// TIA Portal V17 export
// export: Created 2025-07-01T09:58:23.6431093Z, ExportSetting WithDefaults, DisplayName Totally Integrated Automation Portal, DisplayVersion V17 Update 8, DisplayName TIA Portal Openness, DisplayVersion V17 Update 8, DisplayName TIA Portal Version Control Interface, DisplayVersion V17, DisplayName SINAMICS Startdrive Advanced, DisplayVersion V17 SP2, DisplayName SINAMICS Startdrive G110M, G120, G120C, G120D, G120P, G115D, DisplayVersion V17 SP2, DisplayName SINAMICS Startdrive G130, G150, S120, S150, SINAMICS MV, S210, DisplayVersion V17 SP2, DisplayName STEP 7 Professional, DisplayVersion V17 Update 8, DisplayName SINUMERIK ONE STEP 7 Toolbox, DisplayVersion V17 Update 12, DisplayName SINUMERIK ONE PLC Basic Program Plus, DisplayVersion V17 Update 12, DisplayName SINUMERIK 840D sl STEP 7 Toolbox, DisplayVersion V17 Update 12, DisplayName STEP 7 Safety, DisplayVersion V17 Update 6, DisplayName WinCC Advanced, DisplayVersion V17 Update 8
FUNCTION_BLOCK "FB10400_PRESSURE_SENSOR"   // FB10400, LAD
{ S7_Optimized_Access := 'FALSE' }
VERSION : 0.1
// stored: AutoNumber false, IsIECCheckEnabled false, SetENOAutomatically false, UDAEnableTagReadback false
   VAR_INPUT
      SENSOR_VALUE_I : Int;   // SENSOR VALUE INPUT
      STATION_CYCLE_RUNNING : Bool;   // STATION CYCLE RUNNING
   END_VAR
   VAR_OUTPUT
      LOW_PRESSURE_ALARM : Bool;   // ASPIRATION PRESSURE TOO LOW ALARM
      HIGH_PRESSURE_ALARM : Bool;   // ASPIRATION PRESSURE TOO HIGH ALARM
      LOW_PRESSURE_WARNING : Bool;   // ASPIRATION PRESSURE TOO LOW WARNING
      HIGH_PRESSURE_WARNING : Bool;   // ASPIRATION PRESSURE TOO HIGH WARNING
   END_VAR
   VAR DB_SPECIFIC
      HMI : Struct
         HIGH_LIMIT_ALARM_VALUE : Real;   // HIGH LIMIT ALARM VALUE
         HIGH_LIMIT_WARNING_VALUE : Real;   // HIGH LIMIT WARNING VALUE
         LOW_LIMIT_ALARM_VALUE : Real;   // LOW LIMIT ALARM VALUE
         LOW_LIMIT_WARNING_VALUE : Real;   // LOW LIMIT WARNING VALUE
      END_STRUCT;
      SETTINGS : Struct
         NORM_MIN_VAL : Int;   // NORMALIZE MIN VALUE
         NORM_MAX_VAL : Int;   // NORMALIZE MAX VALUE
         SCALE_MIN_VAL : Real;   // SCALE MIN VALUE
         SCALE_MAX_VAL : Real;   // SCALE MAX VALUE
         MUL_VAL : Real;   // MULTIPLY VALUE
         DIV_VAL : Real;   // DIVIDE VALUE
         UNIT_NO : Int;   // UNIT NUMBER
      END_STRUCT;
      OUTPUT : Struct
         PRESSURE_VALUE : Real;   // PRESSURE VALUE
      END_STRUCT;
      INTERNAL : Struct
         NORMALIZED_VALUE : Real;   // NORMALIZED VALUE
         SCALED_VALUE : Real;   // SCALED VALUE
         MULTIPLIED_VALUE : Real;   // MULTIPLIED VALUE
      END_STRUCT;
      ALARMS : Struct
         LOW_PRESSURE_ALARM : Bool;   // ASPIRATION PRESSURE TOO LOW ALARM
         HIGH_PRESSURE_ALARM : Bool;   // ASPIRATION PRESSURE TOO HIGH ALARM
         LOW_PRESSURE_WARNING : Bool;   // ASPIRATION PRESSURE TOO LOW WARNING
         HIGH_PRESSURE_WARNING : Bool;   // ASPIRATION PRESSURE TOO HIGH WARNING
      END_STRUCT;
      TIMERS : Struct
         ASPIRATION_LOW_ALARM_TIMER : TON_TIME;
         ASPIRATION_LOW_WARNING_TIMER : TON_TIME;
         ASPIRATION_HIGH_ALARM_TIMER : TON_TIME;
         ASPIRATION_HIGH_WARNING_TIMER : TON_TIME;
      END_STRUCT;
   END_VAR
   VAR_TEMP
      DB_NUMBER : DInt;   // DB NUMBER
   END_VAR
   VAR_TEMP   // added for the SCL form of the ladder/FBD networks
      _w1 : Bool;
   END_VAR
BEGIN

NETWORK
TITLE = READ INSTANCE DB
      L     DINO;
      +     10#800000;
      T     #DB_NUMBER;


REGION Network 2: PRESSURE VALUE
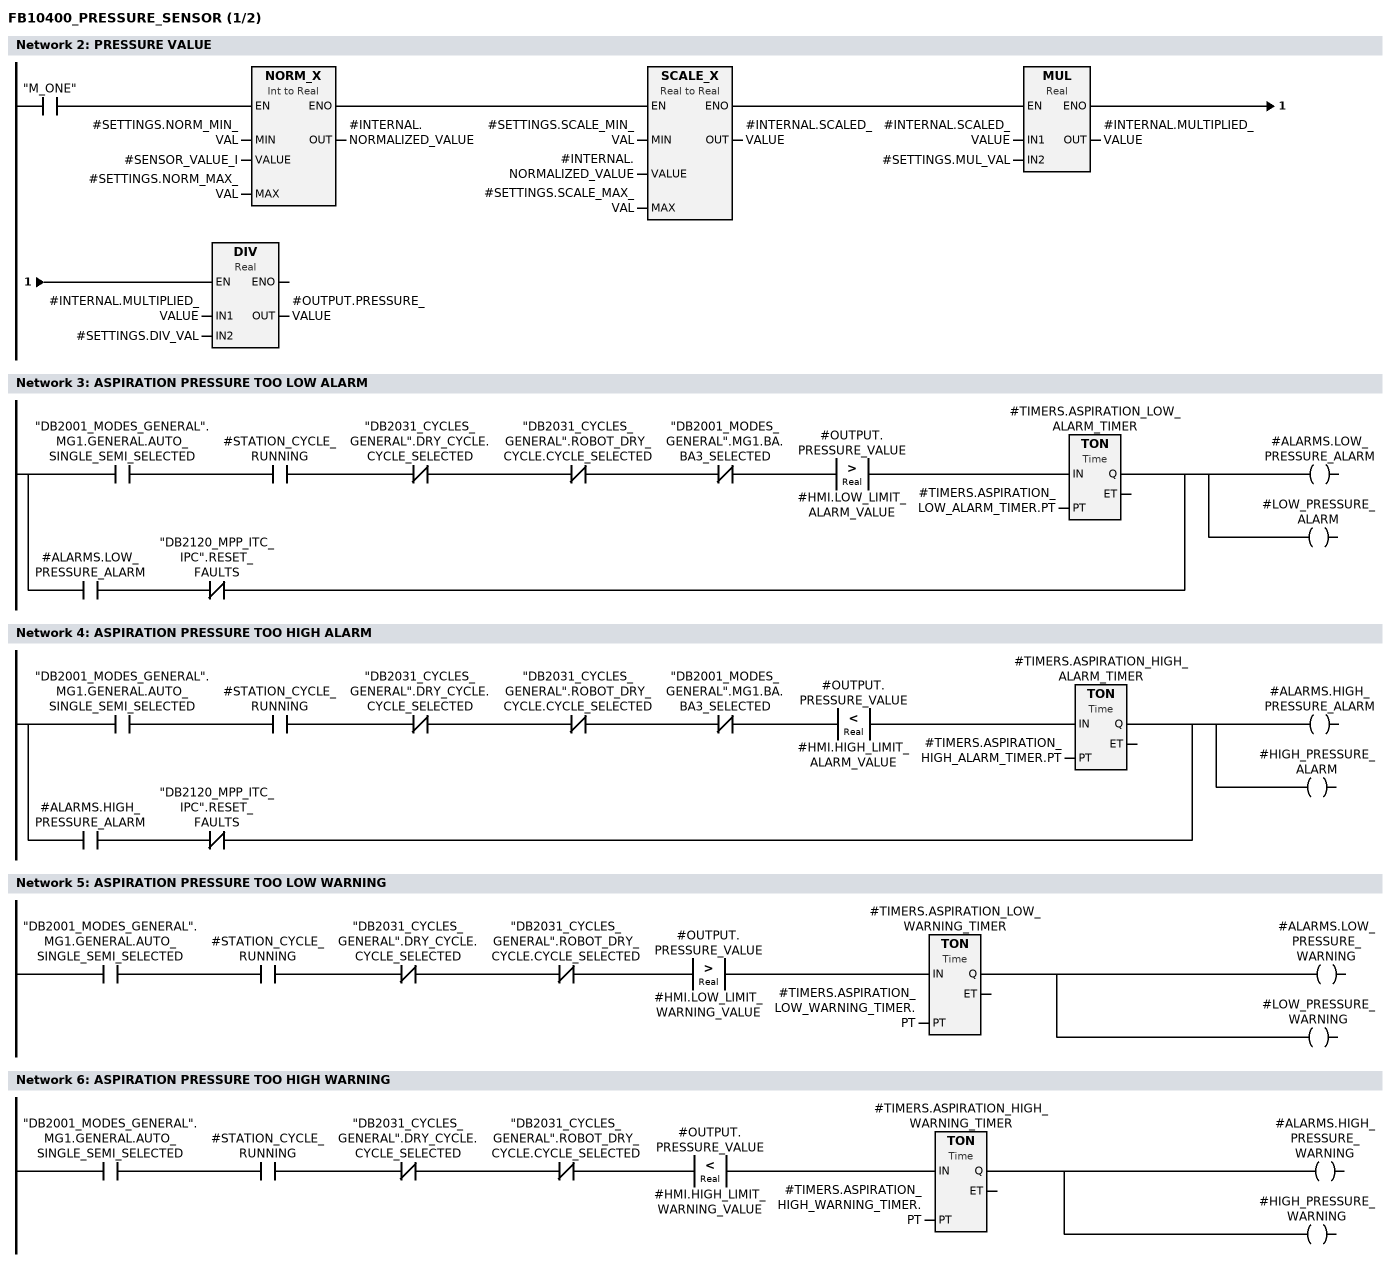
   RUNG wire#powerrail
      Contact( "M_ONE" )
      { S7_Templates := "[SrcType := Int, DestType := Real]" } Normalize(min := #SETTINGS.NORM_MIN_VAL, value := #SENSOR_VALUE_I, max := #SETTINGS.NORM_MAX_VAL, out => #INTERNAL.NORMALIZED_VALUE)
      { S7_Templates := "[SrcType := Real, DestType := Real]" } Scale(min := #SETTINGS.SCALE_MIN_VAL, value := #INTERNAL.NORMALIZED_VALUE, max := #SETTINGS.SCALE_MAX_VAL, out => #INTERNAL.SCALED_VALUE)
      { S7_Templates := "SrcType := Real" } Mul(in1 := #INTERNAL.SCALED_VALUE, in2 := #SETTINGS.MUL_VAL, out => #INTERNAL.MULTIPLIED_VALUE)
      { S7_Templates := "SrcType := Real" } Div(in1 := #INTERNAL.MULTIPLIED_VALUE, in2 := #SETTINGS.DIV_VAL, out => #OUTPUT.PRESSURE_VALUE)
   END_RUNG
   // the same network as SCL:
   IF "M_ONE" THEN
       #INTERNAL.NORMALIZED_VALUE := NORM_X(MIN := #SETTINGS.NORM_MIN_VAL, VALUE := #SENSOR_VALUE_I, MAX := #SETTINGS.NORM_MAX_VAL);
       #INTERNAL.SCALED_VALUE := SCALE_X(MIN := #SETTINGS.SCALE_MIN_VAL, VALUE := #INTERNAL.NORMALIZED_VALUE, MAX := #SETTINGS.SCALE_MAX_VAL);
       #INTERNAL.MULTIPLIED_VALUE := #INTERNAL.SCALED_VALUE * #SETTINGS.MUL_VAL;
       #OUTPUT.PRESSURE_VALUE := #INTERNAL.MULTIPLIED_VALUE / #SETTINGS.DIV_VAL;
   END_IF;
END_REGION

REGION Network 3: ASPIRATION PRESSURE TOO LOW ALARM
   RUNG wire#powerrail
      Contact( "DB2001_MODES_GENERAL".MG1.GENERAL.AUTO_SINGLE_SEMI_SELECTED )
      Contact( #STATION_CYCLE_RUNNING )
      I_Contact( "DB2031_CYCLES_GENERAL".DRY_CYCLE.CYCLE_SELECTED )
      I_Contact( "DB2031_CYCLES_GENERAL".ROBOT_DRY_CYCLE.CYCLE_SELECTED )
      I_Contact( "DB2001_MODES_GENERAL".MG1.BA.BA3_SELECTED )
      { S7_Templates := "SrcType := Real" } GT_Contact(in1 := #OUTPUT.PRESSURE_VALUE, in2 := #HMI.LOW_LIMIT_ALARM_VALUE)
      { S7_Templates := "time_type := Time" } #TIMERS.ASPIRATION_LOW_ALARM_TIMER.TON(pt := #TIMERS.ASPIRATION_LOW_ALARM_TIMER.PT, et =>)
      wire#w1
      Coil( #ALARMS.LOW_PRESSURE_ALARM )
   END_RUNG
   RUNG wire#powerrail
      Contact( #ALARMS.LOW_PRESSURE_ALARM )
      I_Contact( "DB2120_MPP_ITC_IPC".RESET_FAULTS )
   END_RUNG wire#w1
   RUNG wire#w1
      Coil( #LOW_PRESSURE_ALARM )
   END_RUNG
   // the same network as SCL:
   #TIMERS.ASPIRATION_LOW_ALARM_TIMER.TON(IN := "DB2001_MODES_GENERAL".MG1.GENERAL.AUTO_SINGLE_SEMI_SELECTED AND #STATION_CYCLE_RUNNING AND NOT "DB2031_CYCLES_GENERAL".DRY_CYCLE.CYCLE_SELECTED AND NOT "DB2031_CYCLES_GENERAL".ROBOT_DRY_CYCLE.CYCLE_SELECTED AND NOT "DB2001_MODES_GENERAL".MG1.BA.BA3_SELECTED AND (#OUTPUT.PRESSURE_VALUE > #HMI.LOW_LIMIT_ALARM_VALUE),
                           PT := #TIMERS.ASPIRATION_LOW_ALARM_TIMER.PT);
   #ALARMS.LOW_PRESSURE_ALARM := #TIMERS.ASPIRATION_LOW_ALARM_TIMER.Q OR (#ALARMS.LOW_PRESSURE_ALARM AND NOT "DB2120_MPP_ITC_IPC".RESET_FAULTS);
   #LOW_PRESSURE_ALARM := #ALARMS.LOW_PRESSURE_ALARM;
END_REGION

REGION Network 4: ASPIRATION PRESSURE TOO HIGH ALARM
   RUNG wire#powerrail
      Contact( "DB2001_MODES_GENERAL".MG1.GENERAL.AUTO_SINGLE_SEMI_SELECTED )
      Contact( #STATION_CYCLE_RUNNING )
      I_Contact( "DB2031_CYCLES_GENERAL".DRY_CYCLE.CYCLE_SELECTED )
      I_Contact( "DB2031_CYCLES_GENERAL".ROBOT_DRY_CYCLE.CYCLE_SELECTED )
      I_Contact( "DB2001_MODES_GENERAL".MG1.BA.BA3_SELECTED )
      { S7_Templates := "SrcType := Real" } LT_Contact(in1 := #OUTPUT.PRESSURE_VALUE, in2 := #HMI.HIGH_LIMIT_ALARM_VALUE)
      { S7_Templates := "time_type := Time" } #TIMERS.ASPIRATION_HIGH_ALARM_TIMER.TON(pt := #TIMERS.ASPIRATION_HIGH_ALARM_TIMER.PT, et =>)
      wire#w1
      Coil( #ALARMS.HIGH_PRESSURE_ALARM )
   END_RUNG
   RUNG wire#powerrail
      Contact( #ALARMS.HIGH_PRESSURE_ALARM )
      I_Contact( "DB2120_MPP_ITC_IPC".RESET_FAULTS )
   END_RUNG wire#w1
   RUNG wire#w1
      Coil( #HIGH_PRESSURE_ALARM )
   END_RUNG
   // the same network as SCL:
   #TIMERS.ASPIRATION_HIGH_ALARM_TIMER.TON(IN := "DB2001_MODES_GENERAL".MG1.GENERAL.AUTO_SINGLE_SEMI_SELECTED AND #STATION_CYCLE_RUNNING AND NOT "DB2031_CYCLES_GENERAL".DRY_CYCLE.CYCLE_SELECTED AND NOT "DB2031_CYCLES_GENERAL".ROBOT_DRY_CYCLE.CYCLE_SELECTED AND NOT "DB2001_MODES_GENERAL".MG1.BA.BA3_SELECTED AND (#OUTPUT.PRESSURE_VALUE < #HMI.HIGH_LIMIT_ALARM_VALUE),
                           PT := #TIMERS.ASPIRATION_HIGH_ALARM_TIMER.PT);
   #ALARMS.HIGH_PRESSURE_ALARM := #TIMERS.ASPIRATION_HIGH_ALARM_TIMER.Q OR (#ALARMS.HIGH_PRESSURE_ALARM AND NOT "DB2120_MPP_ITC_IPC".RESET_FAULTS);
   #HIGH_PRESSURE_ALARM := #ALARMS.HIGH_PRESSURE_ALARM;
END_REGION

REGION Network 5: ASPIRATION PRESSURE TOO LOW WARNING
   RUNG wire#powerrail
      Contact( "DB2001_MODES_GENERAL".MG1.GENERAL.AUTO_SINGLE_SEMI_SELECTED )
      Contact( #STATION_CYCLE_RUNNING )
      I_Contact( "DB2031_CYCLES_GENERAL".DRY_CYCLE.CYCLE_SELECTED )
      I_Contact( "DB2031_CYCLES_GENERAL".ROBOT_DRY_CYCLE.CYCLE_SELECTED )
      { S7_Templates := "SrcType := Real" } GT_Contact(in1 := #OUTPUT.PRESSURE_VALUE, in2 := #HMI.LOW_LIMIT_WARNING_VALUE)
      { S7_Templates := "time_type := Time" } #TIMERS.ASPIRATION_LOW_WARNING_TIMER.TON(pt := #TIMERS.ASPIRATION_LOW_WARNING_TIMER.PT, et =>)
      wire#w1
      Coil( #ALARMS.LOW_PRESSURE_WARNING )
   END_RUNG
   RUNG wire#w1
      Coil( #LOW_PRESSURE_WARNING )
   END_RUNG
   // the same network as SCL:
   #TIMERS.ASPIRATION_LOW_WARNING_TIMER.TON(IN := "DB2001_MODES_GENERAL".MG1.GENERAL.AUTO_SINGLE_SEMI_SELECTED AND #STATION_CYCLE_RUNNING AND NOT "DB2031_CYCLES_GENERAL".DRY_CYCLE.CYCLE_SELECTED AND NOT "DB2031_CYCLES_GENERAL".ROBOT_DRY_CYCLE.CYCLE_SELECTED AND (#OUTPUT.PRESSURE_VALUE > #HMI.LOW_LIMIT_WARNING_VALUE),
                           PT := #TIMERS.ASPIRATION_LOW_WARNING_TIMER.PT);
   #ALARMS.LOW_PRESSURE_WARNING := #TIMERS.ASPIRATION_LOW_WARNING_TIMER.Q;
   #LOW_PRESSURE_WARNING := #TIMERS.ASPIRATION_LOW_WARNING_TIMER.Q;
END_REGION

REGION Network 6: ASPIRATION PRESSURE TOO HIGH WARNING
   RUNG wire#powerrail
      Contact( "DB2001_MODES_GENERAL".MG1.GENERAL.AUTO_SINGLE_SEMI_SELECTED )
      Contact( #STATION_CYCLE_RUNNING )
      I_Contact( "DB2031_CYCLES_GENERAL".DRY_CYCLE.CYCLE_SELECTED )
      I_Contact( "DB2031_CYCLES_GENERAL".ROBOT_DRY_CYCLE.CYCLE_SELECTED )
      { S7_Templates := "SrcType := Real" } LT_Contact(in1 := #OUTPUT.PRESSURE_VALUE, in2 := #HMI.HIGH_LIMIT_WARNING_VALUE)
      { S7_Templates := "time_type := Time" } #TIMERS.ASPIRATION_HIGH_WARNING_TIMER.TON(pt := #TIMERS.ASPIRATION_HIGH_WARNING_TIMER.PT, et =>)
      wire#w1
      Coil( #ALARMS.HIGH_PRESSURE_WARNING )
   END_RUNG
   RUNG wire#w1
      Coil( #HIGH_PRESSURE_WARNING )
   END_RUNG
   // the same network as SCL:
   #TIMERS.ASPIRATION_HIGH_WARNING_TIMER.TON(IN := "DB2001_MODES_GENERAL".MG1.GENERAL.AUTO_SINGLE_SEMI_SELECTED AND #STATION_CYCLE_RUNNING AND NOT "DB2031_CYCLES_GENERAL".DRY_CYCLE.CYCLE_SELECTED AND NOT "DB2031_CYCLES_GENERAL".ROBOT_DRY_CYCLE.CYCLE_SELECTED AND (#OUTPUT.PRESSURE_VALUE < #HMI.HIGH_LIMIT_WARNING_VALUE),
                           PT := #TIMERS.ASPIRATION_HIGH_WARNING_TIMER.PT);
   #ALARMS.HIGH_PRESSURE_WARNING := #TIMERS.ASPIRATION_HIGH_WARNING_TIMER.Q;
   #HIGH_PRESSURE_WARNING := #TIMERS.ASPIRATION_HIGH_WARNING_TIMER.Q;
END_REGION

REGION Network 7: IMMEDIATE STOP AND STOP END OF CYCLE ALARMS
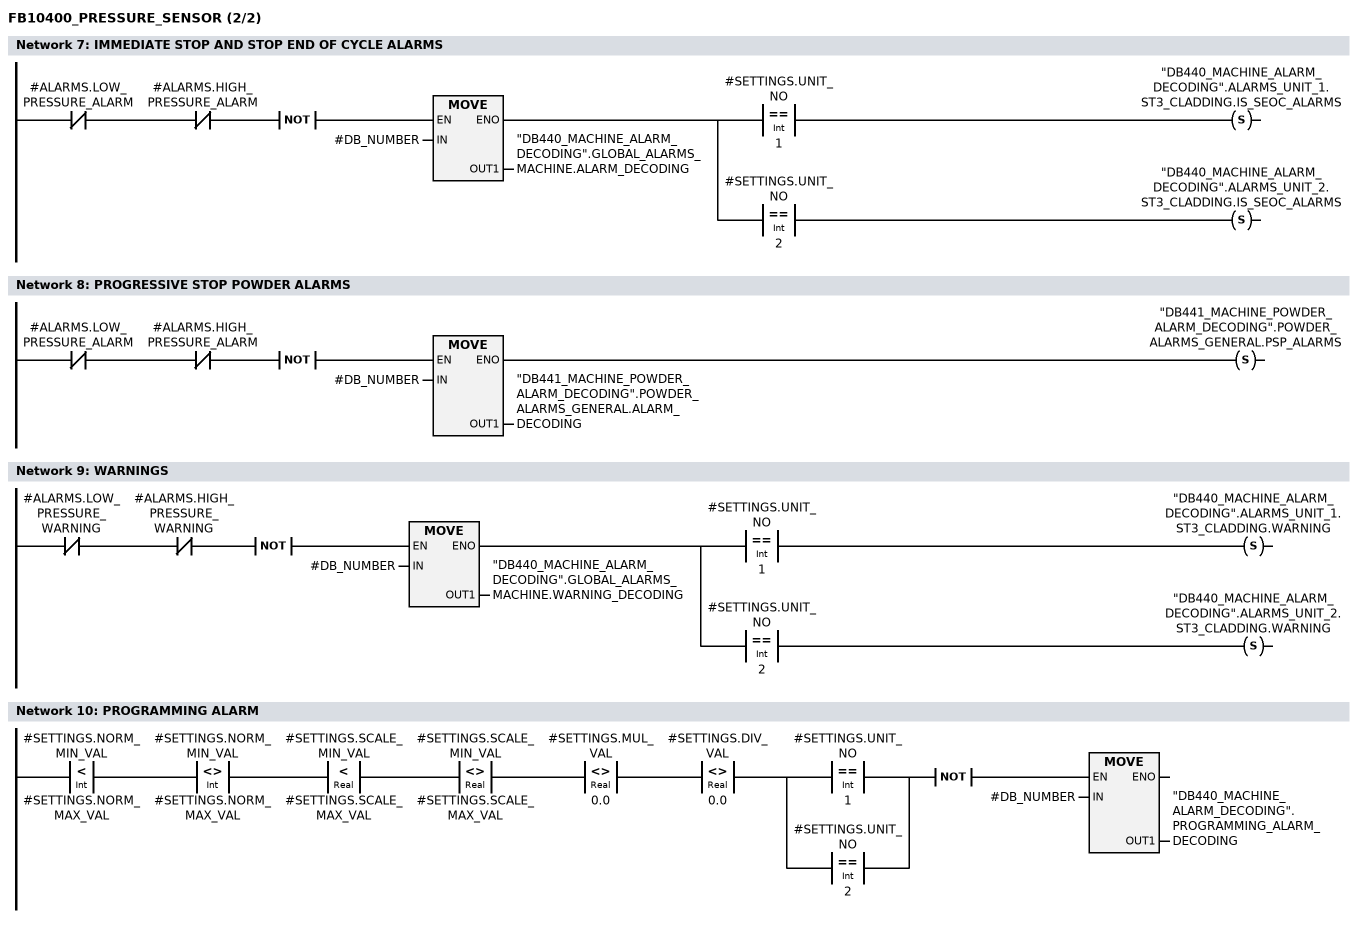
   RUNG wire#powerrail
      I_Contact( #ALARMS.LOW_PRESSURE_ALARM )
      I_Contact( #ALARMS.HIGH_PRESSURE_ALARM )
      Not()
      { S7_GenerateENO := "TRUE" } Move(in := #DB_NUMBER, out1 => "DB440_MACHINE_ALARM_DECODING".GLOBAL_ALARMS_MACHINE.ALARM_DECODING)
      wire#w1
      { S7_Templates := "SrcType := Int" } EQ_Contact(in1 := #SETTINGS.UNIT_NO, in2 := 1)
      S_Coil( "DB440_MACHINE_ALARM_DECODING".ALARMS_UNIT_1.ST3_CLADDING.IS_SEOC_ALARMS )
   END_RUNG
   RUNG wire#w1
      { S7_Templates := "SrcType := Int" } EQ_Contact(in1 := #SETTINGS.UNIT_NO, in2 := 2)
      S_Coil( "DB440_MACHINE_ALARM_DECODING".ALARMS_UNIT_2.ST3_CLADDING.IS_SEOC_ALARMS )
   END_RUNG
   // the same network as SCL:
   // ENO of a box is taken as its EN; it also drops when the box reports an error
   #_w1 := NOT (NOT #ALARMS.LOW_PRESSURE_ALARM AND NOT #ALARMS.HIGH_PRESSURE_ALARM);
   IF #_w1 THEN "DB440_MACHINE_ALARM_DECODING".GLOBAL_ALARMS_MACHINE.ALARM_DECODING := #DB_NUMBER; END_IF;
   IF #_w1 AND (#SETTINGS.UNIT_NO = 1) THEN
       "DB440_MACHINE_ALARM_DECODING".ALARMS_UNIT_1.ST3_CLADDING.IS_SEOC_ALARMS := TRUE;
   END_IF;
   IF #_w1 AND (#SETTINGS.UNIT_NO = 2) THEN
       "DB440_MACHINE_ALARM_DECODING".ALARMS_UNIT_2.ST3_CLADDING.IS_SEOC_ALARMS := TRUE;
   END_IF;
END_REGION

REGION Network 8: PROGRESSIVE STOP POWDER ALARMS
   RUNG wire#powerrail
      I_Contact( #ALARMS.LOW_PRESSURE_ALARM )
      I_Contact( #ALARMS.HIGH_PRESSURE_ALARM )
      Not()
      { S7_GenerateENO := "TRUE" } Move(in := #DB_NUMBER, out1 => "DB441_MACHINE_POWDER_ALARM_DECODING".POWDER_ALARMS_GENERAL.ALARM_DECODING)
      S_Coil( "DB441_MACHINE_POWDER_ALARM_DECODING".POWDER_ALARMS_GENERAL.PSP_ALARMS )
   END_RUNG
   // the same network as SCL:
   // ENO of a box is taken as its EN; it also drops when the box reports an error
   IF NOT (NOT #ALARMS.LOW_PRESSURE_ALARM AND NOT #ALARMS.HIGH_PRESSURE_ALARM) THEN
       "DB441_MACHINE_POWDER_ALARM_DECODING".POWDER_ALARMS_GENERAL.ALARM_DECODING := #DB_NUMBER;
       "DB441_MACHINE_POWDER_ALARM_DECODING".POWDER_ALARMS_GENERAL.PSP_ALARMS := TRUE;
   END_IF;
END_REGION

REGION Network 9: WARNINGS
   RUNG wire#powerrail
      I_Contact( #ALARMS.LOW_PRESSURE_WARNING )
      I_Contact( #ALARMS.HIGH_PRESSURE_WARNING )
      Not()
      Move(in := #DB_NUMBER, out1 => "DB440_MACHINE_ALARM_DECODING".GLOBAL_ALARMS_MACHINE.WARNING_DECODING)
      wire#w1
      { S7_Templates := "SrcType := Int" } EQ_Contact(in1 := #SETTINGS.UNIT_NO, in2 := 1)
      S_Coil( "DB440_MACHINE_ALARM_DECODING".ALARMS_UNIT_1.ST3_CLADDING.WARNING )
   END_RUNG
   RUNG wire#w1
      { S7_Templates := "SrcType := Int" } EQ_Contact(in1 := #SETTINGS.UNIT_NO, in2 := 2)
      S_Coil( "DB440_MACHINE_ALARM_DECODING".ALARMS_UNIT_2.ST3_CLADDING.WARNING )
   END_RUNG
   // the same network as SCL:
   #_w1 := NOT (NOT #ALARMS.LOW_PRESSURE_WARNING AND NOT #ALARMS.HIGH_PRESSURE_WARNING);
   IF #_w1 THEN "DB440_MACHINE_ALARM_DECODING".GLOBAL_ALARMS_MACHINE.WARNING_DECODING := #DB_NUMBER; END_IF;
   IF #_w1 AND (#SETTINGS.UNIT_NO = 1) THEN
       "DB440_MACHINE_ALARM_DECODING".ALARMS_UNIT_1.ST3_CLADDING.WARNING := TRUE;
   END_IF;
   IF #_w1 AND (#SETTINGS.UNIT_NO = 2) THEN
       "DB440_MACHINE_ALARM_DECODING".ALARMS_UNIT_2.ST3_CLADDING.WARNING := TRUE;
   END_IF;
END_REGION

REGION Network 10: PROGRAMMING ALARM
   RUNG wire#powerrail
      { S7_Templates := "SrcType := Int" } LT_Contact(in1 := #SETTINGS.NORM_MIN_VAL, in2 := #SETTINGS.NORM_MAX_VAL)
      { S7_Templates := "SrcType := Int" } NE_Contact(in1 := #SETTINGS.NORM_MIN_VAL, in2 := #SETTINGS.NORM_MAX_VAL)
      { S7_Templates := "SrcType := Real" } LT_Contact(in1 := #SETTINGS.SCALE_MIN_VAL, in2 := #SETTINGS.SCALE_MAX_VAL)
      { S7_Templates := "SrcType := Real" } NE_Contact(in1 := #SETTINGS.SCALE_MIN_VAL, in2 := #SETTINGS.SCALE_MAX_VAL)
      { S7_Templates := "SrcType := Real" } NE_Contact(in1 := #SETTINGS.MUL_VAL, in2 := 0.0)
      { S7_Templates := "SrcType := Real" } NE_Contact(in1 := #SETTINGS.DIV_VAL, in2 := 0.0)
      wire#w1
      { S7_Templates := "SrcType := Int" } EQ_Contact(in1 := #SETTINGS.UNIT_NO, in2 := 1)
      wire#w2
      Not()
      Move(in := #DB_NUMBER, out1 => "DB440_MACHINE_ALARM_DECODING".PROGRAMMING_ALARM_DECODING)
   END_RUNG
   RUNG wire#w1
      { S7_Templates := "SrcType := Int" } EQ_Contact(in1 := #SETTINGS.UNIT_NO, in2 := 2)
   END_RUNG wire#w2
   // the same network as SCL:
   IF NOT ((#SETTINGS.NORM_MIN_VAL < #SETTINGS.NORM_MAX_VAL) AND (#SETTINGS.NORM_MIN_VAL <> #SETTINGS.NORM_MAX_VAL) AND (#SETTINGS.SCALE_MIN_VAL < #SETTINGS.SCALE_MAX_VAL) AND (#SETTINGS.SCALE_MIN_VAL <> #SETTINGS.SCALE_MAX_VAL) AND (#SETTINGS.MUL_VAL <> 0.0) AND (#SETTINGS.DIV_VAL <> 0.0) AND ((#SETTINGS.UNIT_NO = 1) OR (#SETTINGS.UNIT_NO = 2))) THEN
       "DB440_MACHINE_ALARM_DECODING".PROGRAMMING_ALARM_DECODING := #DB_NUMBER;
   END_IF;
END_REGION
END_FUNCTION_BLOCK
